TYPE "PosFbk_RTN"
VERSION : 0.1
// Block: PosFbk_RTN
   STRUCT
      Preset : Struct
         Pulses : DInt;
         Units : LReal;
      END_STRUCT;
      Config : Struct
         Resolution : LReal;
      END_STRUCT;
   END_STRUCT;

END_TYPE
